FUNCTION_BLOCK KeyValueCollectionChangedEventHandler EXTENDS KeyValueCollectionEventHandler

METHOD PUBLIC HandleEvent
VAR_INPUT
	Event : I_Event;
END_VAR
VAR
	changedEvent : I_KeyValueCollectionChangedEvent;
END_VAR
IF __QUERYINTERFACE(Event, changedEvent) THEN
	_eventReceived := TRUE;
	fromExpected := changedEvent.Target = expectedOriginator;
END_IF
END_METHOD

END_FUNCTION_BLOCK

(* stored: Version 1.1.0.1, ProductVersion 3.1.4024.12
   POU KeyValueCollectionChangedEventHandler: Id {bd953192-5868-4092-b0e7-29bdcae5445c}, SpecialFunc None
   Method HandleEvent: Id {1002c501-7dd7-4e38-b142-e1836c898162} *)
